FUNCTION_BLOCK FB_ExecutorCutX EXTENDS FB_ExecutorBase
VAR
    // Zostawiasz tu TYLKO to, co dotyczy bezpośrednio osi X!
    _AxisX          : SPT_Motion_Control.I_BasicAxis;
    _AxisY          : SPT_Motion_Control.I_BasicAxis;
    _AxisZ          : SPT_Motion_Control.I_BasicAxis;
    _Cylinder       : I_Cylinder;                     
    _RecipeBuilder  : I_RecipeBuilder;
    _Config         : REFERENCE TO ST_GantryXYZ_Config;
END_VAR

PROPERTY AxisX : I_BasicAxis
GET
AxisX := _AxisX;
END_GET
SET
_AxisX := AxisX;
END_SET
END_PROPERTY

PROPERTY AxisY : I_BasicAxis
GET
AxisY := _AxisY;
END_GET
SET
_AxisY := AxisY;
END_SET
END_PROPERTY

PROPERTY AxisZ : I_BasicAxis
GET
AxisZ := _AxisZ;
END_GET
SET
_AxisZ := AxisZ;
END_SET
END_PROPERTY

PROPERTY Config : REFERENCE TO ST_GantryXYZ_Config
GET
Config REF= _Config;
END_GET
SET
_Config REF= Config;
END_SET
END_PROPERTY

METHOD PUBLIC  CyclicLogic
VAR_INST
    // Lokalne zmienne pomocnicze na czas trwania cyklu
    localSegmentsCutX : ARRAY[1..32] OF ST_CutSegment;
    currentSeg        : ST_CutSegment;
END_VAR

StepTimer();


// Zabezpieczenie na wypadek braku wstrzykniętych referencji!
IF _RecipeBuilder = 0 OR NOT __ISVALIDREF(_Config) THEN
    Trace('Brak referencji w ExecutorCutX!');
    RETURN;
END_IF

// 1. Zrzut całej tablicy z Właściwości (Property) do zmiennej lokalnej
localSegmentsCutX := _RecipeBuilder.SegmentsCutX;

IF iCurrentSegment < 1 THEN iCurrentSegment := 1; END_IF
IF iCurrentSegment > 32 THEN iCurrentSegment := 32; END_IF

// 2. Wyciągnięcie konkretnego segmentu dla aktualnego kroku
// (Bezpieczny odczyt z lokalnej pamięci)
currentSeg := localSegmentsCutX[iCurrentSegment];

CASE nStep OF
	
	0: // IDLE - maszyna czeka na wywołanie Execute()

    // -------- Inicjalizacja --------
    5:
        IF _AxisX.Enable() AND _AxisY.Enable() AND _AxisZ.Enable() THEN
            
            Trace('SegmentExecutionX Started');
            IF _RecipeBuilder.SegmentsToCutX <= 0 THEN
                nStep := 1000; // Nie ma czego ciąć, zakończ natychmiast
                RETURN;
            END_IF;

            // Jednorazowe nastawy dynamiki z wstrzykniętej konfiguracji
            _AxisX.Acceleration := 500;   _AxisX.Deceleration := 8000;
            _AxisY.Acceleration := 500;   _AxisY.Deceleration := 8000;
            _AxisZ.Acceleration := 500;   _AxisZ.Deceleration := 8000;
            
            _AxisX.Velocity := _Config.RapidSpeedX;
            _AxisY.Velocity := _Config.RapidSpeedY;
            _AxisZ.Velocity := _Config.RapidSpeedZ;

            iCurrentSegment := 1;
            
            IF NOT _AxisX.Busy AND NOT _AxisY.Busy AND NOT _AxisZ.Busy THEN
                nStep := 10;
            END_IF     
        END_IF

    // -------- Dojazd do początku cięcia --------
    10:
        _AxisX.MoveAbsolute(
            _RecipeBuilder.SegmentsCutX[iCurrentSegment].Start.X + _Config.CutterXOffsetX + _Config.GlobalOffset, 
            0);
        _AxisY.MoveAbsolute(
            _RecipeBuilder.SegmentsCutX[iCurrentSegment].Start.Y + _Config.CutterXOffsetY + _Config.GlobalOffset, 
            0);
        nStep := 20;

    20: // Czekamy na pozycję XY
        IF _AxisX.InPosition AND _AxisY.InPosition THEN 
            nStep := 30;
        END_IF

    // -------- Wysunięcie siłownika (Ostrze w dół) --------
    30:
        _Cylinder.Extend();
        nStep := 40;

    40: 
        IF _Cylinder.Extended THEN
            // Zmiana prędkości na roboczą z konfiguracji
            _AxisX.Velocity := _Config.CuttingSpeedX;
            _AxisY.Velocity := _Config.CuttingSpeedY;
            nStep := 50;
        END_IF
            
    50: // Czekanie (Cutting Idle Time)
        StepTimer(IN := TRUE, PT := REAL_TO_TIME(_Config.CuttingIdleTime * 1000.0));
        IF StepTimer.Q THEN
            StepTimer(IN := FALSE); // Reset timera na przyszłość
            nStep := 60;
        END_IF

    // -------- Cięcie XY do końca odcinka --------
    60:
        _AxisX.MoveAbsolute(
            _RecipeBuilder.SegmentsCutX[iCurrentSegment].Stop.X + _Config.CutterXOffsetX + _Config.GlobalOffset, 
            0);
        _AxisY.MoveAbsolute(
            _RecipeBuilder.SegmentsCutX[iCurrentSegment].Stop.Y + _Config.CutterXOffsetY + _Config.GlobalOffset, 
            0);
        nStep := 70;

    70: // Czekamy na koniec cięcia
        IF _AxisX.InPosition AND _AxisY.InPosition THEN
            nStep := 80;
        END_IF

    // -------- Chowanie ostrza i przygotowanie następnego --------
    80:
        _Cylinder.Retract();
        nStep := 85;

    85: 
        IF _Cylinder.Retracted THEN
             iCurrentSegment := iCurrentSegment + 1; 
             nStep := 90;
        END_IF    

    90: // Drugi Idle Time
        StepTimer(IN := TRUE, PT := REAL_TO_TIME(_Config.CuttingIdleTime * 1000.0));
        IF StepTimer.Q THEN
            StepTimer(IN := FALSE);
            
            // Powrót do prędkości dojazdowej
            _AxisX.Velocity := _Config.RapidSpeedX;
            _AxisY.Velocity := _Config.RapidSpeedY;
            
            IF iCurrentSegment > _RecipeBuilder.SegmentsToCutX THEN
                nStep := 1000; // Koniec wszystkich segmentów
            ELSE
                nStep := 10;   // Skok do następnego odcinka
            END_IF
        END_IF

    // -------- Zakończenie pracy Executora --------
1000:
        Trace('SegmentExecutionX-FINISHED');
        _bBusy := FALSE; // Wyłączamy flagę pracy
        _bDone := TRUE;  // Dajemy sygnał Orchestratorowi, że skończyliśmy!
        nStep := 0;      // Wracamy do stanu IDLE

        
END_CASE
END_METHOD

PROPERTY Cylinder : I_Cylinder
GET
Cylinder := _Cylinder;
END_GET
SET
_Cylinder := Cylinder;
END_SET
END_PROPERTY

PROPERTY RecipeBuilder : I_RecipeBuilder
GET
RecipeBuilder := _RecipeBuilder;
END_GET
SET
_RecipeBuilder := RecipeBuilder;
END_SET
END_PROPERTY

END_FUNCTION_BLOCK

(* stored: Version 1.1.0.1, ProductVersion 3.1.4024.15
   POU FB_ExecutorCutX: Id {91737efa-f775-4890-9334-f282750ffd75}, SpecialFunc None
   Property AxisX: Id {bf7bf1e8-4628-46ee-9a7f-8b243677db34}
   Get Get: Id {d93144b5-dd29-483a-8b76-9038e49c9a6d}
   Set Set: Id {7ab3348b-b4bb-4d6b-bd39-8185e257a35e}
   Property AxisY: Id {d6d2cedb-0eda-4e75-a191-4d8ce3a9bbf4}
   Get Get: Id {3b91612c-9793-4f68-8ba4-cfcfaf6d0685}
   Set Set: Id {cefe518b-6ed4-4e66-9928-cc421068c6b9}
   Property AxisZ: Id {411509dc-9082-4584-89ca-2ff1afd18787}
   Get Get: Id {3ef8d70c-0902-4da9-8ae9-200f5cfec13c}
   Set Set: Id {fbb69cdf-dc2f-457b-88ac-db5f43779a82}
   Property Config: Id {d4eaeb02-3324-4dfb-bb21-b43618bd8a51}
   Get Get: Id {b1b19422-708f-4729-8a80-0ec5c4e56462}
   Set Set: Id {855da8aa-c381-42d4-945c-30bcec476610}
   Method CyclicLogic: Id {49e00514-3bc2-4f55-9abc-aaedafe38071}
   Property Cylinder: Id {0546bd86-401b-41c0-a683-bbe302146fdd}
   Get Get: Id {622de191-a52d-4efd-af87-b0787b5827c2}
   Set Set: Id {f831b18a-1816-415a-82f6-5aeacd4161b5}
   Property RecipeBuilder: Id {cbbaad3b-7e73-402c-b55d-1c46460bfd77}
   Get Get: Id {ee8216eb-1e0d-45e3-8dfd-22bbcbfa2526}
   Set Set: Id {1d93da46-a542-4ef2-b525-3599ad0c4f6e} *)
